{attribute 'GeneratedUsingTerminal: EL6090-0000-0016'}
{attribute addProperty BoxType "EL6090-0000-0016"}
{attribute addProperty Id "UpBOOL1DownBOOL1LeftBOOL1RightBOOL1EnterBOOL1TxPDO_ToggleBOOL1"}
{attribute addProperty CRC "3823631634"}
{attribute addProperty Size "6"}
TYPE Status_E3E7FD12 :
STRUCT
	{attribute addProperty Name "Up"}
	Up : BOOL;
	{attribute addProperty Name "Down"}
	Down : BOOL;
	{attribute addProperty Name "Left"}
	Left : BOOL;
	{attribute addProperty Name "Right"}
	Right : BOOL;
	{attribute addProperty Name "Enter"}
	Enter : BOOL;
	{attribute addProperty Name "TxPDO_Toggle"}
	TxPDO_Toggle : BOOL;
END_STRUCT
END_TYPE

(* stored: Version 1.2.0.0, ProductVersion 3.1.4024.9
   DUT Status_E3E7FD12: Id {030c78e5-5e4c-49ef-a8c7-90f6c7475ecb} *)
